// TIA Portal V16 export
// export: Created 2021-09-08T12:46:09.5319372Z, ExportSetting WithDefaults, DisplayName Totally Integrated Automation Portal, DisplayVersion V16 Update 3, DisplayName TIA Portal Version Control Interface, DisplayVersion V16 Update 2, DisplayName TIA Portal Openness, DisplayVersion V16 Update 3, DisplayName TIA Portal Teamcenter Gateway, DisplayVersion V16, DisplayName STEP 7 Professional, DisplayVersion V16 Update 3, DisplayName STEP 7 Safety, DisplayVersion V16, DisplayName WinCC Advanced, DisplayVersion V16 Update 3
FUNCTION "setState" : Void   // FC3, FBD
{ S7_Optimized_Access := 'TRUE' }
VERSION : 0.1
// stored: AutoNumber true, IsIECCheckEnabled false, SetENOAutomatically false, UDAEnableTagReadback false
   VAR_INPUT
      condition : Bool;
      hexVal : Word;
   END_VAR
   VAR_IN_OUT
      state : Word;
   END_VAR
BEGIN

REGION Network 1 (SCL)
   IF #condition THEN
       // Statement section IF
       #state := #state OR #hexVal;
   ELSE
       #state := #state AND NOT #hexVal;
   END_IF;
END_REGION
END_FUNCTION
